{attribute 'qualified_only'}
{attribute 'strict'}
{attribute 'to_string'}
TYPE ST170_RFID_e :
(
    RESET := 0, // Reset

    INIT := 100, // Initialisieren 
    Init_vertical_homing,
    Init_vertical_down,

    READY := 999,  // READY to Start, Init Done 
    START := 1000, // Start Zyklisch

    waitOnMover,     // wait until the mover is there
    MOVER_NEEDED_OP, // Since here, a mover in position is needed to perform the action

    vertical_up,         // 
    RFID_start,    // 
    RFID_wait_on_result, // 
    RFID_read,     // 
    vertical_down,       // 

    SYNC_MOVER_LEAVE, // MoverMan need to take the mover
    MOVER_FREE_OP,       // Ab here, operation without mover can be done

    DONE := 8000,  // Ablauf beendet 
    ERROR := 9000, // Fehler 
    _max
);
END_TYPE

(* stored: Version 1.1.0.1, ProductVersion 3.1.4024.6
   EnumerationTextList ST170_RFID_e: Id {a4cb59e1-b76d-41d7-bf84-e550b73cc65f} *)
